FUNCTION_BLOCK fbWaitBlock IMPLEMENTS IWaitBlock
VAR_INPUT
END_VAR
VAR_OUTPUT
END_VAR
VAR
END_VAR

END_FUNCTION_BLOCK

(* stored: Version 1.1.0.1, ProductVersion 3.1.4024.6
   POU fbWaitBlock: Id {b5ed8a97-d186-41dd-948c-47796c432afe}, SpecialFunc None *)
